FUNCTION_BLOCK TLController (* Composite Function Block Type *)
  (* Standard: 61499-2 *)
  (* Version 0.2, 2003-12-05, JHC, Rockwell Automation, Renamed from NEWCOMPFB. *)
  (* Version 0.1, 2002-01-08, JHC, Rockwell Automation, Added DLY FB as example. *)
  (* Version 0.0, 2000-05-27, JHC, Rockwell Automation *)
  (* Compiler header: package fb.rt.template; *)
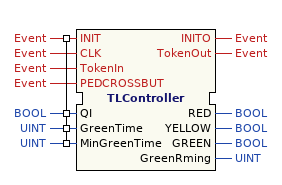
  EVENT_INPUT
    INIT WITH QI, GreenTime, MinGreenTime; (* Initialization Request *)
    CLK;
    TokenIn;
    PEDCROSSBUT;
  END_EVENT
  EVENT_OUTPUT
    INITO; (* Initialization Confirm *)
    TokenOut;
  END_EVENT
  VAR_INPUT
    QI : BOOL; (* Input event qualifier *)
    GreenTime : UINT;
    MinGreenTime : UINT;
  END_VAR
  VAR_OUTPUT
    RED : BOOL;
    YELLOW : BOOL;
    GREEN : BOOL;
    GreenRming : UINT;
  END_VAR
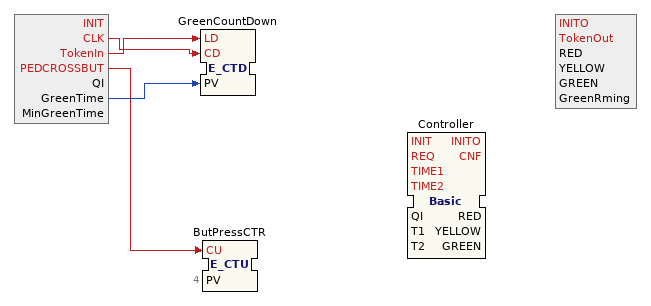
  FBS
    GreenCountDown : E_CTD;
    ButPressCTR : E_CTU(PV := 4);
    Controller : Basic;
  END_FBS
  EVENT_CONNECTIONS
    TokenIn TO GreenCountDown.LD;
    PEDCROSSBUT TO ButPressCTR.CU;
    CLK TO GreenCountDown.CD;
  END_CONNECTIONS
  DATA_CONNECTIONS
    GreenTime TO GreenCountDown.PV;
  END_CONNECTIONS
END_FUNCTION_BLOCK
